INTERFACE I_FileHandler EXTENDS ZigasLibs_Core.I_FileProperties, ZigasLibs_Core.I_RequiresAmsAddress

// Creates the file. Returns TRUE when done - method needs to be called until it returns TRUE!
METHOD Create : BOOL
VAR_INPUT
	bOverwrite	: BOOL;	// If file already exists, it will be deleted and crated once again (content will be lost!)
END_VAR
END_METHOD

// Deletes the file, if it exists. Returns TRUE when done - method needs to be called until it returns TRUE!
METHOD Delete : BOOL
END_METHOD

// Gets the error state, if any of the functions failed.
PROPERTY Error : BOOL
GET
END_GET
END_PROPERTY

// Checks if the file exists. Returns TRUE when done - method needs to be called until it returns TRUE!
METHOD Exists : BOOL
VAR_INPUT
	refFileExists	: REFERENCE TO BOOL;	// When mehod is finished, the variable provided here will have the result, TRUE if file exists, FALSE if not.
END_VAR
END_METHOD

// Reads the content of the opened file to the target buffer.
// Returns TRUE when done - method needs to be called until it returns TRUE!
METHOD Read : BOOL
VAR_INPUT
	buffer	: ANY;
END_VAR
END_METHOD

METHOD Reset
VAR_INPUT
END_VAR
END_METHOD

// Writes the content to the end of the file (appends).
// Returns TRUE when done - method needs to be called until it returns TRUE!
METHOD WriteBinary_Append : BOOL
VAR_INPUT
	data	: ANY;
END_VAR
END_METHOD

// Writes the content to the the file (overwrites any existing content).
// Returns TRUE when done - method needs to be called until it returns TRUE!
METHOD WriteBinary_Overwrite : BOOL
VAR_INPUT
	data	: ANY;
END_VAR
END_METHOD

// Writes the string content to the end of the file (appends). If the file does not exist, it will be created.
// Returns TRUE when done - method needs to be called until it returns TRUE!
METHOD WriteLine_Append : BOOL
VAR_INPUT
	sContent	: Tc2_System.T_MaxString;	// Text to be written.
END_VAR
END_METHOD

// Writes the string content to file and overwrites any existing content. If the file does not exist, it will be created.
// Returns TRUE when done - method needs to be called until it returns TRUE!
METHOD WriteLine_Overwrite : BOOL
VAR_INPUT
	sContent	: Tc2_System.T_MaxString;	// Text to be written.
END_VAR
END_METHOD

END_INTERFACE

(* stored: Version 1.1.0.1, ProductVersion 3.1.4024.13
   Itf I_FileHandler: Id {4b78af44-5cd0-09b9-35c8-80b3588f1952}
   Method Create: Id {17e79720-8695-0d8d-1a43-b288c2f2e7b5}
   Method Delete: Id {c90accf8-2301-0d95-25eb-c6db2c0a8bd7}
   Property Error: Id {5fddca4c-4791-0235-1001-725d1b007e34}
   Get Get: Id {150a6457-4279-0493-37e2-eae3f023eafc}
   Method Exists: Id {8bdd038a-9abc-04cb-3144-e5aef79c2eb4}
   Method Read: Id {9c7915fb-0cde-0641-0546-30c103dec798}
   Method Reset: Id {8831fa7d-53e9-07aa-3fa5-54b2380ecff6}
   Method WriteBinary_Append: Id {b12151c7-19f1-0487-35c3-7d39348a832f}
   Method WriteBinary_Overwrite: Id {b797a373-2575-086a-0c90-2cab40d8d804}
   Method WriteLine_Append: Id {a7d31bb1-3d2e-0774-2e5b-de4112925f65}
   Method WriteLine_Overwrite: Id {0f47c073-4a01-0770-238b-441ab0b7e38a} *)
